// TIA Portal V18 export
// export: Created 2025-12-01T12:38:33.9724391Z, ExportSetting None, DisplayName Totally Integrated Automation Portal, DisplayVersion V18 Update 5, DisplayName TIA Portal Openness, DisplayVersion V18 Update 5, DisplayName TIA Portal Teamcenter Gateway, DisplayVersion V18, DisplayName TIA Portal Version Control Interface, DisplayVersion V18, DisplayName STEP 7 Professional, DisplayVersion V18 Update 5, DisplayName STEP 7 Safety, DisplayVersion V18, DisplayName WinCC Professional, DisplayVersion V18 Update 5
FUNCTION "ST10Cyl_interface61-70" : Void   // FC1026, LAD
{ S7_Optimized_Access := 'FALSE' }
// stored: AutoNumber false, SetENOAutomatically false
   VAR_INPUT
      AlwaysON : Bool;
      E_stop : Bool;
   END_VAR
   VAR_TEMP
      tTest : Bool;
   END_VAR
BEGIN

REGION Network 1 (SCL): Cylinder 61-70 IO Interface (SCL)
   (*
   //Cylinder61 IO  K-reserveLifting3LiftingCylinder
   //Input
   "ST10Cylinder".Cy[61].In.WorkPositionSensor := "iK-reserveLifting3LiftingCylinderInWP";
   "ST10Cylinder".Cy[61].In.HomePositionSensor := "iK-reserveLifting3LiftingCylinderInHP";
   //Output
   "oK-reserveLifting3LiftingCylinderToWP" := "ST10Cylinder".Cy[61].Out.GoWorkPosition;
   "oK-reserveLifting3LiftingCylinderToHP" := "ST10Cylinder".Cy[61].Out.GoHomePosition;

   //Cylinder62 IO  K-reserveLifting3PalletLocationCylinder
   //Input
   "ST10Cylinder".Cy[62].In.WorkPositionSensor := "iK-reserveLifting3PalletLocationCylinderInWP";
   "ST10Cylinder".Cy[62].In.HomePositionSensor := "iK-reserveLifting3PalletLocationCylinderInHP";
   //Output
   "oK-reserveLifting3PalletLocationCylinderToWP" := "ST10Cylinder".Cy[62].Out.GoWorkPosition;
   "oK-reserveLifting3PalletLocationCylinderToHP" := "ST10Cylinder".Cy[62].Out.GoHomePosition;

   //Cylinder63 IO  K-reserveLoadingStopperCylinder1_1
   //Input
   "ST10Cylinder".Cy[63].In.WorkPositionSensor := "oK-reserveLoadingStopperCylinder1_1";
   "ST10Cylinder".Cy[63].In.HomePositionSensor := NOT "oK-reserveLoadingStopperCylinder1_1";
   //Output
   "oK-reserveLoadingStopperCylinder1_1" := "ST10Cylinder".Cy[63].Out.GoWorkPosition;
   //"oI-0030TrayLoading6trayStopperCylinderToHP" := "ST10Cylinder".Cy[63].Out.GoHomePosition;

   //Cylinder64 IO  K-reserveLoadingStopperCylinder1_2
   //Input
   "ST10Cylinder".Cy[64].In.WorkPositionSensor := "oK-reserveLoadingStopperCylinder1_2";
   "ST10Cylinder".Cy[64].In.HomePositionSensor := NOT "oK-reserveLoadingStopperCylinder1_2";
   //Output
   "oK-reserveLoadingStopperCylinder1_2" := "ST10Cylinder".Cy[64].Out.GoWorkPosition;
   //"oI-0060TrayLoadingTaketrayCylinderToHP" := "ST10Cylinder".Cy[64].Out.GoHomePosition;

   //Cylinder65 IO  K-reserveLoadingStopperCylinder2_1
   //Input
   "ST10Cylinder".Cy[65].In.WorkPositionSensor := "oK-reserveLoadingStopperCylinder2_1";
   "ST10Cylinder".Cy[65].In.HomePositionSensor := NOT "oK-reserveLoadingStopperCylinder2_1";
   //Output
   "oK-reserveLoadingStopperCylinder2_1" := "ST10Cylinder".Cy[65].Out.GoWorkPosition;
   //"oI-0050TrayLoadingTrayCylinderToHP" := "ST10Cylinder".Cy[65].Out.GoHomePosition;

   //Cylinder66 K-reserveLoadingStopperCylinder2_2
   //Input
   "ST10Cylinder".Cy[66].In.WorkPositionSensor := "oK-reserveLoadingStopperCylinder2_2";
   "ST10Cylinder".Cy[66].In.HomePositionSensor := NOT "oK-reserveLoadingStopperCylinder2_2";
   //Output
   "oK-reserveLoadingStopperCylinder2_2" := "ST10Cylinder".Cy[66].Out.GoWorkPosition;
   //"oI-0060TrayLoadingTraySupportCylinder1ToHP" := "ST10Cylinder".Cy[66].Out.GoHomePosition;

   //Cylinder67 K-reserveLoadingStopperCylinder3_1
   //Input
   "ST10Cylinder".Cy[67].In.WorkPositionSensor := "oK-reserveLoadingStopperCylinder3_1";
   "ST10Cylinder".Cy[67].In.HomePositionSensor := NOT "oK-reserveLoadingStopperCylinder3_1";
   //Output
   "oK-reserveLoadingStopperCylinder3_1" := "ST10Cylinder".Cy[67].Out.GoWorkPosition;
   //"oI-0070TrayLoadingTraySupportCylinder6ToHP" := "ST10Cylinder".Cy[67].Out.GoHomePosition;

   //Cylinder68 K-reserveLoadingStopperCylinder3_2
   //Input
   "ST10Cylinder".Cy[68].In.WorkPositionSensor := "oK-reserveLoadingStopperCylinder3_2";
   "ST10Cylinder".Cy[68].In.HomePositionSensor := NOT "oK-reserveLoadingStopperCylinder3_2";
   //Output
   "oK-reserveLoadingStopperCylinder3_2" := "ST10Cylinder".Cy[68].Out.GoWorkPosition;
   //"oI-0080TrayLoadingTrayLocationCylinderToHP" := "ST10Cylinder".Cy[68].Out.GoHomePosition;

   //Cylinder69 K-reserveLoadingStopperCylinder4_1
   //Input
   "ST10Cylinder".Cy[69].In.WorkPositionSensor := "oK-reserveLoadingStopperCylinder4_1";
   "ST10Cylinder".Cy[69].In.HomePositionSensor := NOT "oK-reserveLoadingStopperCylinder4_1";
   //Output
   "oK-reserveLoadingStopperCylinder4_1" := "ST10Cylinder".Cy[69].Out.GoWorkPosition;
   //"oI-0090TrayLoadingTrayUnloadingLiftingCylinderToHP" := "ST10Cylinder".Cy[69].Out.GoHomePosition;

   //Cylinder70 K-reserveLoadingStopperCylinder4_2
   // //Input
   "ST10Cylinder".Cy[70].In.WorkPositionSensor := "oK-reserveLoadingStopperCylinder4_2";
   "ST10Cylinder".Cy[70].In.HomePositionSensor := NOT "oK-reserveLoadingStopperCylinder4_2";
   // //Output
   "oK-reserveLoadingStopperCylinder4_2" := "ST10Cylinder".Cy[70].Out.GoWorkPosition;
   // "Feeding washer  lift Cylinder ToHP" := "ST10Cylinder".Cy[70].Out.GoHomePosition;
   *)
END_REGION

REGION Network 2: CY61 interface K-reserveLifting3LiftingCylinder
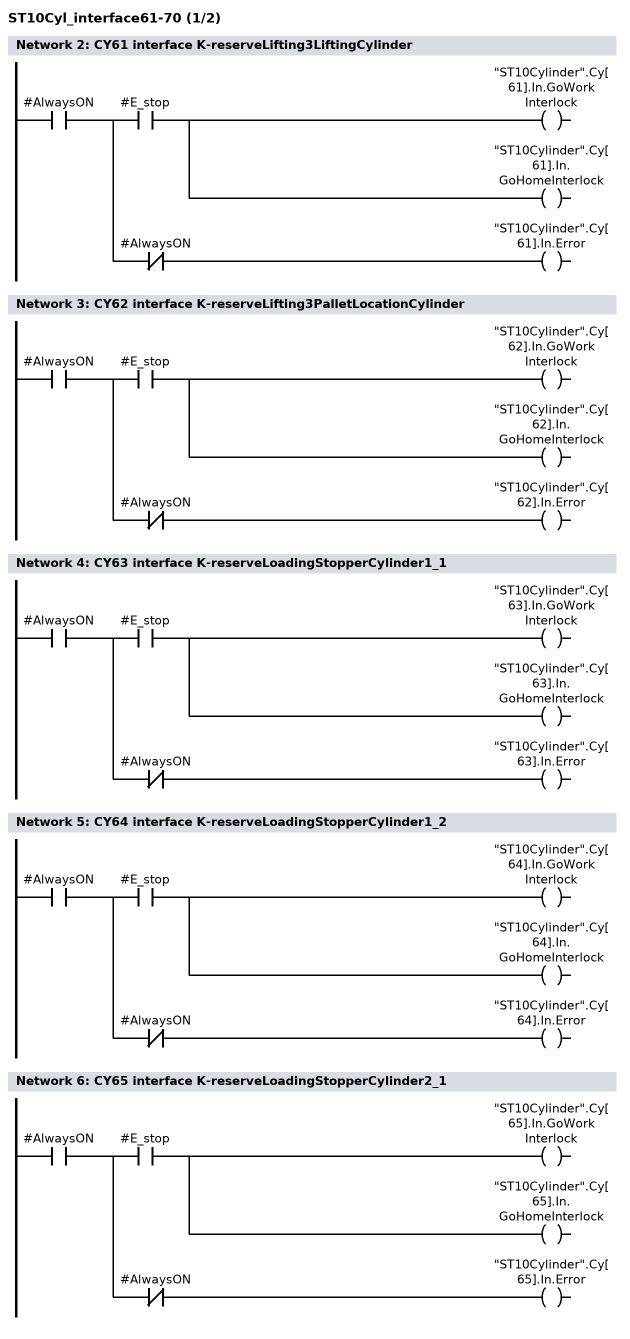
   RUNG wire#powerrail
      Contact( #AlwaysON )
      wire#w1
      Contact( #E_stop )
      wire#w2
      Coil( "ST10Cylinder".Cy[61].In.GoWorkInterlock )
   END_RUNG
   RUNG wire#w2
      Coil( "ST10Cylinder".Cy[61].In.GoHomeInterlock )
   END_RUNG
   RUNG wire#w1
      I_Contact( #AlwaysON )
      Coil( "ST10Cylinder".Cy[61].In.Error )
   END_RUNG
   // the same network as SCL:
   "ST10Cylinder".Cy[61].In.GoWorkInterlock := #AlwaysON AND #E_stop;
   "ST10Cylinder".Cy[61].In.GoHomeInterlock := #AlwaysON AND #E_stop;
   "ST10Cylinder".Cy[61].In.Error := #AlwaysON AND NOT #AlwaysON;
END_REGION

REGION Network 3: CY62 interface K-reserveLifting3PalletLocationCylinder
   RUNG wire#powerrail
      Contact( #AlwaysON )
      wire#w1
      Contact( #E_stop )
      wire#w2
      Coil( "ST10Cylinder".Cy[62].In.GoWorkInterlock )
   END_RUNG
   RUNG wire#w2
      Coil( "ST10Cylinder".Cy[62].In.GoHomeInterlock )
   END_RUNG
   RUNG wire#w1
      I_Contact( #AlwaysON )
      Coil( "ST10Cylinder".Cy[62].In.Error )
   END_RUNG
   // the same network as SCL:
   "ST10Cylinder".Cy[62].In.GoWorkInterlock := #AlwaysON AND #E_stop;
   "ST10Cylinder".Cy[62].In.GoHomeInterlock := #AlwaysON AND #E_stop;
   "ST10Cylinder".Cy[62].In.Error := #AlwaysON AND NOT #AlwaysON;
END_REGION

REGION Network 4: CY63 interface K-reserveLoadingStopperCylinder1_1
   RUNG wire#powerrail
      Contact( #AlwaysON )
      wire#w1
      Contact( #E_stop )
      wire#w2
      Coil( "ST10Cylinder".Cy[63].In.GoWorkInterlock )
   END_RUNG
   RUNG wire#w2
      Coil( "ST10Cylinder".Cy[63].In.GoHomeInterlock )
   END_RUNG
   RUNG wire#w1
      I_Contact( #AlwaysON )
      Coil( "ST10Cylinder".Cy[63].In.Error )
   END_RUNG
   // the same network as SCL:
   "ST10Cylinder".Cy[63].In.GoWorkInterlock := #AlwaysON AND #E_stop;
   "ST10Cylinder".Cy[63].In.GoHomeInterlock := #AlwaysON AND #E_stop;
   "ST10Cylinder".Cy[63].In.Error := #AlwaysON AND NOT #AlwaysON;
END_REGION

REGION Network 5: CY64 interface K-reserveLoadingStopperCylinder1_2
   RUNG wire#powerrail
      Contact( #AlwaysON )
      wire#w1
      Contact( #E_stop )
      wire#w2
      Coil( "ST10Cylinder".Cy[64].In.GoWorkInterlock )
   END_RUNG
   RUNG wire#w2
      Coil( "ST10Cylinder".Cy[64].In.GoHomeInterlock )
   END_RUNG
   RUNG wire#w1
      I_Contact( #AlwaysON )
      Coil( "ST10Cylinder".Cy[64].In.Error )
   END_RUNG
   // the same network as SCL:
   "ST10Cylinder".Cy[64].In.GoWorkInterlock := #AlwaysON AND #E_stop;
   "ST10Cylinder".Cy[64].In.GoHomeInterlock := #AlwaysON AND #E_stop;
   "ST10Cylinder".Cy[64].In.Error := #AlwaysON AND NOT #AlwaysON;
END_REGION

REGION Network 6: CY65 interface K-reserveLoadingStopperCylinder2_1
   RUNG wire#powerrail
      Contact( #AlwaysON )
      wire#w1
      Contact( #E_stop )
      wire#w2
      Coil( "ST10Cylinder".Cy[65].In.GoWorkInterlock )
   END_RUNG
   RUNG wire#w2
      Coil( "ST10Cylinder".Cy[65].In.GoHomeInterlock )
   END_RUNG
   RUNG wire#w1
      I_Contact( #AlwaysON )
      Coil( "ST10Cylinder".Cy[65].In.Error )
   END_RUNG
   // the same network as SCL:
   "ST10Cylinder".Cy[65].In.GoWorkInterlock := #AlwaysON AND #E_stop;
   "ST10Cylinder".Cy[65].In.GoHomeInterlock := #AlwaysON AND #E_stop;
   "ST10Cylinder".Cy[65].In.Error := #AlwaysON AND NOT #AlwaysON;
END_REGION

REGION Network 7: CY66 interface K-reserveLoadingStopperCylinder2_2
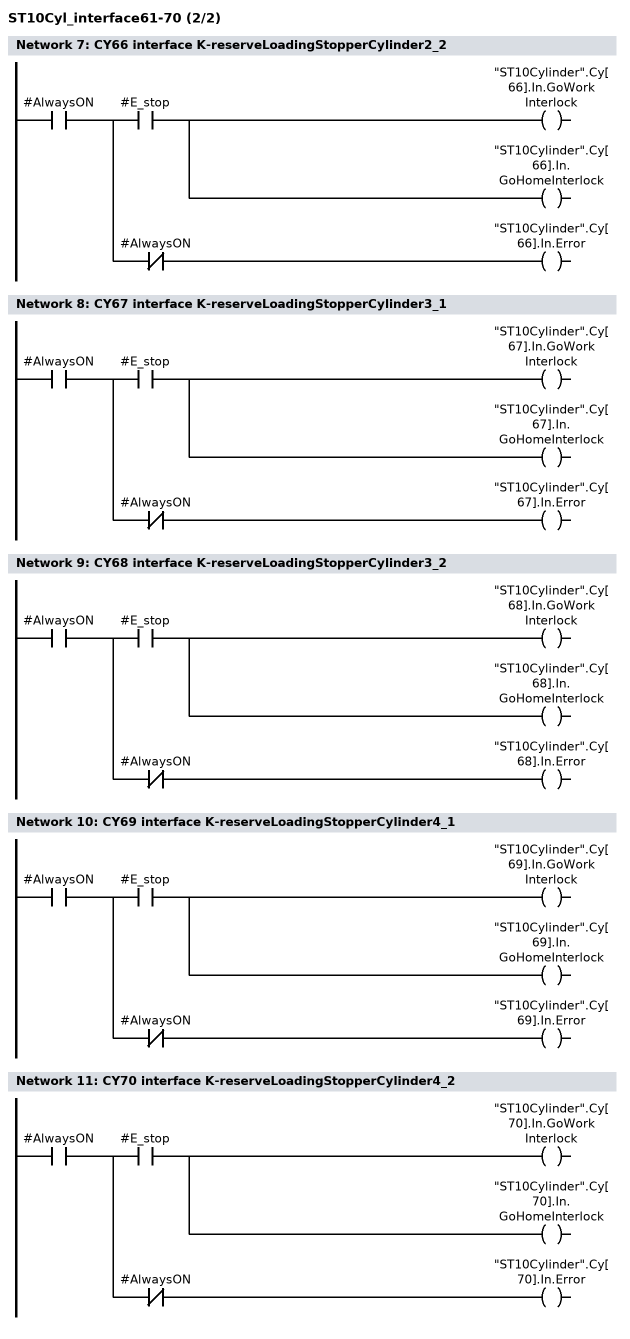
   RUNG wire#powerrail
      Contact( #AlwaysON )
      wire#w1
      Contact( #E_stop )
      wire#w2
      Coil( "ST10Cylinder".Cy[66].In.GoWorkInterlock )
   END_RUNG
   RUNG wire#w2
      Coil( "ST10Cylinder".Cy[66].In.GoHomeInterlock )
   END_RUNG
   RUNG wire#w1
      I_Contact( #AlwaysON )
      Coil( "ST10Cylinder".Cy[66].In.Error )
   END_RUNG
   // the same network as SCL:
   "ST10Cylinder".Cy[66].In.GoWorkInterlock := #AlwaysON AND #E_stop;
   "ST10Cylinder".Cy[66].In.GoHomeInterlock := #AlwaysON AND #E_stop;
   "ST10Cylinder".Cy[66].In.Error := #AlwaysON AND NOT #AlwaysON;
END_REGION

REGION Network 8: CY67 interface K-reserveLoadingStopperCylinder3_1
   RUNG wire#powerrail
      Contact( #AlwaysON )
      wire#w1
      Contact( #E_stop )
      wire#w2
      Coil( "ST10Cylinder".Cy[67].In.GoWorkInterlock )
   END_RUNG
   RUNG wire#w2
      Coil( "ST10Cylinder".Cy[67].In.GoHomeInterlock )
   END_RUNG
   RUNG wire#w1
      I_Contact( #AlwaysON )
      Coil( "ST10Cylinder".Cy[67].In.Error )
   END_RUNG
   // the same network as SCL:
   "ST10Cylinder".Cy[67].In.GoWorkInterlock := #AlwaysON AND #E_stop;
   "ST10Cylinder".Cy[67].In.GoHomeInterlock := #AlwaysON AND #E_stop;
   "ST10Cylinder".Cy[67].In.Error := #AlwaysON AND NOT #AlwaysON;
END_REGION

REGION Network 9: CY68 interface K-reserveLoadingStopperCylinder3_2
   RUNG wire#powerrail
      Contact( #AlwaysON )
      wire#w1
      Contact( #E_stop )
      wire#w2
      Coil( "ST10Cylinder".Cy[68].In.GoWorkInterlock )
   END_RUNG
   RUNG wire#w2
      Coil( "ST10Cylinder".Cy[68].In.GoHomeInterlock )
   END_RUNG
   RUNG wire#w1
      I_Contact( #AlwaysON )
      Coil( "ST10Cylinder".Cy[68].In.Error )
   END_RUNG
   // the same network as SCL:
   "ST10Cylinder".Cy[68].In.GoWorkInterlock := #AlwaysON AND #E_stop;
   "ST10Cylinder".Cy[68].In.GoHomeInterlock := #AlwaysON AND #E_stop;
   "ST10Cylinder".Cy[68].In.Error := #AlwaysON AND NOT #AlwaysON;
END_REGION

REGION Network 10: CY69 interface K-reserveLoadingStopperCylinder4_1
   RUNG wire#powerrail
      Contact( #AlwaysON )
      wire#w1
      Contact( #E_stop )
      wire#w2
      Coil( "ST10Cylinder".Cy[69].In.GoWorkInterlock )
   END_RUNG
   RUNG wire#w2
      Coil( "ST10Cylinder".Cy[69].In.GoHomeInterlock )
   END_RUNG
   RUNG wire#w1
      I_Contact( #AlwaysON )
      Coil( "ST10Cylinder".Cy[69].In.Error )
   END_RUNG
   // the same network as SCL:
   "ST10Cylinder".Cy[69].In.GoWorkInterlock := #AlwaysON AND #E_stop;
   "ST10Cylinder".Cy[69].In.GoHomeInterlock := #AlwaysON AND #E_stop;
   "ST10Cylinder".Cy[69].In.Error := #AlwaysON AND NOT #AlwaysON;
END_REGION

REGION Network 11: CY70 interface K-reserveLoadingStopperCylinder4_2
   RUNG wire#powerrail
      Contact( #AlwaysON )
      wire#w1
      Contact( #E_stop )
      wire#w2
      Coil( "ST10Cylinder".Cy[70].In.GoWorkInterlock )
   END_RUNG
   RUNG wire#w2
      Coil( "ST10Cylinder".Cy[70].In.GoHomeInterlock )
   END_RUNG
   RUNG wire#w1
      I_Contact( #AlwaysON )
      Coil( "ST10Cylinder".Cy[70].In.Error )
   END_RUNG
   // the same network as SCL:
   "ST10Cylinder".Cy[70].In.GoWorkInterlock := #AlwaysON AND #E_stop;
   "ST10Cylinder".Cy[70].In.GoHomeInterlock := #AlwaysON AND #E_stop;
   "ST10Cylinder".Cy[70].In.Error := #AlwaysON AND NOT #AlwaysON;
END_REGION
END_FUNCTION
